(* IEC 61131-3 sources: NVM-AquaFeed-Platform/02_Software_Design/PLC/07_Implementation/Function_Blocks, 14 files *)

(* ---- FB_AlarmManager.st ---- *)
FUNCTION_BLOCK FB_AlarmManager
VAR_INPUT
    astConditions : ARRAY[0..31] OF ST_AlarmCondition;

    xAcknowledgeRequest : BOOL;
    xResetRequest : BOOL;
    udiCommandSequence : UDINT;
    uiTargetAlarmCode : UINT;
    eTargetSource : E_AlarmSource;
    usiTargetLineId : USINT;
    uiTargetDeviceId : UINT;

    udiAcceptedEventSequence : UDINT;
END_VAR
VAR_OUTPUT
    astActiveAlarms : ARRAY[0..63] OF ST_Alarm;
    stPendingEvent : ST_AlarmEvent;
    xPendingEventValid : BOOL;
    uiPendingEventCount : UINT;

    xAnyAlarmActive : BOOL;
    xAnyBlockingAlarm : BOOL;
    xAnyCriticalAlarm : BOOL;
    xAnyEmergencyAlarm : BOOL;
    eHighestSeverity : E_AlarmSeverity;
    uiActiveAlarmCount : UINT;

    xTableOverflow : BOOL;
    xEventBufferOverflow : BOOL;
    xInputRejected : BOOL;
    uiInputResultCode : UINT;

    xCommandAccepted : BOOL;
    xCommandRejected : BOOL;
    uiCommandResultCode : UINT;
    udiLastProcessedCommandSequence : UDINT;
END_VAR
VAR
    astEventBuffer : ARRAY[0..127] OF ST_AlarmEvent;
    uiEventReadIndex : UINT;
    uiEventWriteIndex : UINT;
    udiEventSequence : UDINT;
    xHasProcessedCommand : BOOL;

    iCondition : INT;
    iPreviousCondition : INT;
    iAlarm : INT;
    iFoundAlarm : INT;
    iFreeAlarm : INT;
    iCommandAlarm : INT;

    xDefinitionValid : BOOL;
    xSeverityValid : BOOL;
    xDuplicateUpdate : BOOL;
    xPolicyMatches : BOOL;
    xEmitEvent : BOOL;
    eEmitEventType : E_AlarmEventType;
END_VAR
VAR CONSTANT
    c_uiInputResultNone : UINT := 0;
    c_uiInputResultInvalidDefinition : UINT := 10;
    c_uiInputResultDuplicateKey : UINT := 11;
    c_uiInputResultPolicyChanged : UINT := 12;
    c_uiInputResultTableFull : UINT := 13;

    c_uiCommandResultNone : UINT := 0;
    c_uiCommandResultAccepted : UINT := 1;
    c_uiCommandResultConflict : UINT := 40;
    c_uiCommandResultNotFound : UINT := 41;
    c_uiCommandResultConditionActive : UINT := 42;
    c_uiCommandResultResetNotRequired : UINT := 43;
END_VAR

xCommandAccepted := FALSE;
xCommandRejected := FALSE;
uiCommandResultCode := c_uiCommandResultNone;
xInputRejected := FALSE;
uiInputResultCode := c_uiInputResultNone;

(* Desktop may remove only the exact oldest retained event. *)
IF (uiPendingEventCount > 0) AND
   (udiAcceptedEventSequence <> 0) AND
   (udiAcceptedEventSequence =
    astEventBuffer[uiEventReadIndex].EventSequence) THEN
    IF uiEventReadIndex >= 127 THEN
        uiEventReadIndex := 0;
    ELSE
        uiEventReadIndex := uiEventReadIndex + 1;
    END_IF;
    uiPendingEventCount := uiPendingEventCount - 1;
END_IF;

(* Process at most 32 explicit condition updates in array order. *)
FOR iCondition := 0 TO 31 DO
    IF astConditions[iCondition].Valid THEN
        xDuplicateUpdate := FALSE;
        IF iCondition > 0 THEN
            FOR iPreviousCondition := 0 TO iCondition - 1 DO
                IF astConditions[iPreviousCondition].Valid AND
                   (astConditions[iPreviousCondition].AlarmCode =
                    astConditions[iCondition].AlarmCode) AND
                   (astConditions[iPreviousCondition].Source =
                    astConditions[iCondition].Source) AND
                   (astConditions[iPreviousCondition].LineId =
                    astConditions[iCondition].LineId) AND
                   (astConditions[iPreviousCondition].DeviceId =
                    astConditions[iCondition].DeviceId) THEN
                    xDuplicateUpdate := TRUE;
                END_IF;
            END_FOR;
        END_IF;

        xSeverityValid := FALSE;
        CASE astConditions[iCondition].Severity OF
            ALARM_INFORMATION,
            ALARM_WARNING,
            ALARM_FAULT,
            ALARM_CRITICAL,
            ALARM_EMERGENCY:
                xSeverityValid := TRUE;
        END_CASE;

        xDefinitionValid := xSeverityValid AND
                            (astConditions[iCondition].AlarmCode >= 1000) AND
                            (astConditions[iCondition].AlarmCode <= 1999) AND
                            NOT ((astConditions[iCondition].Severity =
                                  ALARM_INFORMATION) AND
                                 astConditions[iCondition].Blocking);

        IF xDefinitionValid THEN
            CASE astConditions[iCondition].Source OF
                ALARM_SOURCE_SYSTEM:
                    xDefinitionValid :=
                        ((astConditions[iCondition].AlarmCode >= 1000) AND
                         (astConditions[iCondition].AlarmCode <= 1099)) OR
                        ((astConditions[iCondition].AlarmCode >= 1900) AND
                         (astConditions[iCondition].AlarmCode <= 1999));
                ALARM_SOURCE_COMMUNICATION:
                    xDefinitionValid :=
                        ((astConditions[iCondition].AlarmCode >= 1100) AND
                         (astConditions[iCondition].AlarmCode <= 1199)) OR
                        ((astConditions[iCondition].AlarmCode >= 1900) AND
                         (astConditions[iCondition].AlarmCode <= 1999));
                ALARM_SOURCE_SELECTOR:
                    xDefinitionValid :=
                        (astConditions[iCondition].AlarmCode >= 1200) AND
                        (astConditions[iCondition].AlarmCode <= 1299);
                ALARM_SOURCE_BLOWER:
                    xDefinitionValid :=
                        (astConditions[iCondition].AlarmCode >= 1300) AND
                        (astConditions[iCondition].AlarmCode <= 1399);
                ALARM_SOURCE_DOSING:
                    xDefinitionValid :=
                        (astConditions[iCondition].AlarmCode >= 1400) AND
                        (astConditions[iCondition].AlarmCode <= 1499);
                ALARM_SOURCE_LINE:
                    xDefinitionValid :=
                        (astConditions[iCondition].AlarmCode >= 1500) AND
                        (astConditions[iCondition].AlarmCode <= 1599);
                ALARM_SOURCE_SAFETY,
                ALARM_SOURCE_IO:
                    xDefinitionValid :=
                        ((astConditions[iCondition].AlarmCode >= 1600) AND
                         (astConditions[iCondition].AlarmCode <= 1699)) OR
                        ((astConditions[iCondition].Source =
                          ALARM_SOURCE_IO) AND
                         (astConditions[iCondition].AlarmCode >= 1900) AND
                         (astConditions[iCondition].AlarmCode <= 1999));
                ALARM_SOURCE_POWER:
                    xDefinitionValid :=
                        (astConditions[iCondition].AlarmCode >= 1700) AND
                        (astConditions[iCondition].AlarmCode <= 1799);
                ALARM_SOURCE_AUXILIARY:
                    xDefinitionValid :=
                        (astConditions[iCondition].AlarmCode >= 1800) AND
                        (astConditions[iCondition].AlarmCode <= 1899);
            ELSE
                xDefinitionValid := FALSE;
            END_CASE;
        END_IF;

        IF xDuplicateUpdate THEN
            xInputRejected := TRUE;
            uiInputResultCode := c_uiInputResultDuplicateKey;
        ELSIF NOT xDefinitionValid THEN
            xInputRejected := TRUE;
            uiInputResultCode := c_uiInputResultInvalidDefinition;
        ELSE
            iFoundAlarm := -1;
            iFreeAlarm := -1;
            FOR iAlarm := 0 TO 63 DO
                IF (astActiveAlarms[iAlarm].AlarmCode =
                    astConditions[iCondition].AlarmCode) AND
                   (astActiveAlarms[iAlarm].Source =
                    astConditions[iCondition].Source) AND
                   (astActiveAlarms[iAlarm].LineId =
                    astConditions[iCondition].LineId) AND
                   (astActiveAlarms[iAlarm].DeviceId =
                    astConditions[iCondition].DeviceId) THEN
                    iFoundAlarm := iAlarm;
                END_IF;
                IF (iFreeAlarm < 0) AND
                   (astActiveAlarms[iAlarm].State =
                    ALARM_INACTIVE) THEN
                    iFreeAlarm := iAlarm;
                END_IF;
            END_FOR;

            xEmitEvent := FALSE;

            IF astConditions[iCondition].ConditionActive THEN
                IF iFoundAlarm < 0 THEN
                    IF iFreeAlarm < 0 THEN
                        xTableOverflow := TRUE;
                        xInputRejected := TRUE;
                        uiInputResultCode :=
                            c_uiInputResultTableFull;
                    ELSE
                        IF (astActiveAlarms[iFreeAlarm].AlarmCode <>
                            astConditions[iCondition].AlarmCode) OR
                           (astActiveAlarms[iFreeAlarm].Source <>
                            astConditions[iCondition].Source) OR
                           (astActiveAlarms[iFreeAlarm].LineId <>
                            astConditions[iCondition].LineId) OR
                           (astActiveAlarms[iFreeAlarm].DeviceId <>
                            astConditions[iCondition].DeviceId) THEN
                            astActiveAlarms[iFreeAlarm].OccurrenceCount := 0;
                        END_IF;
                        iFoundAlarm := iFreeAlarm;
                    END_IF;
                END_IF;

                IF iFoundAlarm >= 0 THEN
                    xPolicyMatches :=
                        (astActiveAlarms[iFoundAlarm].State =
                         ALARM_INACTIVE) OR
                        ((astActiveAlarms[iFoundAlarm].Severity =
                          astConditions[iCondition].Severity) AND
                         (astActiveAlarms[iFoundAlarm].ResetRequired =
                          astConditions[iCondition].ResetRequired) AND
                         (astActiveAlarms[iFoundAlarm].Blocking =
                          astConditions[iCondition].Blocking));

                    IF NOT xPolicyMatches THEN
                        xInputRejected := TRUE;
                        uiInputResultCode :=
                            c_uiInputResultPolicyChanged;
                    ELSIF astActiveAlarms[iFoundAlarm].State =
                          ALARM_INACTIVE THEN
                        astActiveAlarms[iFoundAlarm].AlarmCode :=
                            astConditions[iCondition].AlarmCode;
                        astActiveAlarms[iFoundAlarm].Source :=
                            astConditions[iCondition].Source;
                        astActiveAlarms[iFoundAlarm].Severity :=
                            astConditions[iCondition].Severity;
                        astActiveAlarms[iFoundAlarm].State :=
                            ALARM_ACTIVE_UNACKNOWLEDGED;
                        astActiveAlarms[iFoundAlarm].LineId :=
                            astConditions[iCondition].LineId;
                        astActiveAlarms[iFoundAlarm].DeviceId :=
                            astConditions[iCondition].DeviceId;
                        astActiveAlarms[iFoundAlarm].ConditionActive := TRUE;
                        astActiveAlarms[iFoundAlarm].Acknowledged := FALSE;
                        astActiveAlarms[iFoundAlarm].ResetRequired :=
                            astConditions[iCondition].ResetRequired;
                        astActiveAlarms[iFoundAlarm].Blocking :=
                            astConditions[iCondition].Blocking;
                        IF astActiveAlarms[iFoundAlarm].OccurrenceCount <
                           65535 THEN
                            astActiveAlarms[iFoundAlarm].OccurrenceCount :=
                                astActiveAlarms[iFoundAlarm].OccurrenceCount + 1;
                        END_IF;
                        xEmitEvent := TRUE;
                        eEmitEventType := ALARM_EVENT_ACTIVATED;
                    ELSE
                        astActiveAlarms[iFoundAlarm].ConditionActive := TRUE;
                    END_IF;
                END_IF;
            ELSE
                IF (iFoundAlarm >= 0) AND
                   (astActiveAlarms[iFoundAlarm].State <>
                    ALARM_INACTIVE) THEN
                    xPolicyMatches :=
                        (astActiveAlarms[iFoundAlarm].Severity =
                         astConditions[iCondition].Severity) AND
                        (astActiveAlarms[iFoundAlarm].ResetRequired =
                         astConditions[iCondition].ResetRequired) AND
                        (astActiveAlarms[iFoundAlarm].Blocking =
                         astConditions[iCondition].Blocking);

                    IF NOT xPolicyMatches THEN
                        xInputRejected := TRUE;
                        uiInputResultCode :=
                            c_uiInputResultPolicyChanged;
                    ELSIF astActiveAlarms[iFoundAlarm].ConditionActive THEN
                        astActiveAlarms[iFoundAlarm].ConditionActive := FALSE;
                        IF astActiveAlarms[iFoundAlarm].ResetRequired THEN
                            astActiveAlarms[iFoundAlarm].State :=
                                ALARM_CLEARED_WAIT_RESET;
                        ELSE
                            astActiveAlarms[iFoundAlarm].State :=
                                ALARM_INACTIVE;
                            astActiveAlarms[iFoundAlarm].Acknowledged := FALSE;
                        END_IF;
                        xEmitEvent := TRUE;
                        eEmitEventType := ALARM_EVENT_CLEARED;
                    END_IF;
                END_IF;
            END_IF;

            IF xEmitEvent AND (iFoundAlarm >= 0) THEN
                IF udiEventSequence >= c_udiCounterMaximum THEN
                    xEventBufferOverflow := TRUE;
                ELSE
                    udiEventSequence := udiEventSequence + 1;
                    astActiveAlarms[iFoundAlarm].EventSequence :=
                        udiEventSequence;
                    IF eEmitEventType = ALARM_EVENT_ACTIVATED THEN
                        astActiveAlarms[iFoundAlarm].ActivationSequence :=
                            udiEventSequence;
                    END_IF;

                    IF uiPendingEventCount >=
                       c_uiAlarmEventCapacity THEN
                        xEventBufferOverflow := TRUE;
                    ELSE
                        astEventBuffer[uiEventWriteIndex].EventSequence :=
                            udiEventSequence;
                        astEventBuffer[uiEventWriteIndex].EventType :=
                            eEmitEventType;
                        astEventBuffer[uiEventWriteIndex].AlarmCode :=
                            astActiveAlarms[iFoundAlarm].AlarmCode;
                        astEventBuffer[uiEventWriteIndex].Source :=
                            astActiveAlarms[iFoundAlarm].Source;
                        astEventBuffer[uiEventWriteIndex].Severity :=
                            astActiveAlarms[iFoundAlarm].Severity;
                        astEventBuffer[uiEventWriteIndex].State :=
                            astActiveAlarms[iFoundAlarm].State;
                        astEventBuffer[uiEventWriteIndex].LineId :=
                            astActiveAlarms[iFoundAlarm].LineId;
                        astEventBuffer[uiEventWriteIndex].DeviceId :=
                            astActiveAlarms[iFoundAlarm].DeviceId;
                        IF uiEventWriteIndex >= 127 THEN
                            uiEventWriteIndex := 0;
                        ELSE
                            uiEventWriteIndex := uiEventWriteIndex + 1;
                        END_IF;
                        uiPendingEventCount := uiPendingEventCount + 1;
                    END_IF;
                END_IF;
            END_IF;
        END_IF;
    END_IF;
END_FOR;

(* Process one idempotent lifecycle command. *)
IF (xAcknowledgeRequest OR xResetRequest) AND
   (NOT xHasProcessedCommand OR
    (udiCommandSequence <>
     udiLastProcessedCommandSequence)) THEN
    udiLastProcessedCommandSequence := udiCommandSequence;
    xHasProcessedCommand := TRUE;
    iCommandAlarm := -1;

    IF xAcknowledgeRequest AND xResetRequest THEN
        xCommandRejected := TRUE;
        uiCommandResultCode := c_uiCommandResultConflict;
    ELSE
        FOR iAlarm := 0 TO 63 DO
            IF (astActiveAlarms[iAlarm].State <>
                ALARM_INACTIVE) AND
               (astActiveAlarms[iAlarm].AlarmCode =
                uiTargetAlarmCode) AND
               (astActiveAlarms[iAlarm].Source =
                eTargetSource) AND
               (astActiveAlarms[iAlarm].LineId =
                usiTargetLineId) AND
               (astActiveAlarms[iAlarm].DeviceId =
                uiTargetDeviceId) THEN
                iCommandAlarm := iAlarm;
            END_IF;
        END_FOR;

        IF iCommandAlarm < 0 THEN
            xCommandRejected := TRUE;
            uiCommandResultCode := c_uiCommandResultNotFound;
        ELSIF xAcknowledgeRequest THEN
            xCommandAccepted := TRUE;
            uiCommandResultCode := c_uiCommandResultAccepted;
            xEmitEvent := FALSE;
            IF NOT astActiveAlarms[iCommandAlarm].Acknowledged THEN
                astActiveAlarms[iCommandAlarm].Acknowledged := TRUE;
                IF astActiveAlarms[iCommandAlarm].State =
                   ALARM_ACTIVE_UNACKNOWLEDGED THEN
                    astActiveAlarms[iCommandAlarm].State :=
                        ALARM_ACTIVE_ACKNOWLEDGED;
                END_IF;
                xEmitEvent := TRUE;
                eEmitEventType := ALARM_EVENT_ACKNOWLEDGED;
            END_IF;
        ELSE
            xEmitEvent := FALSE;
            IF astActiveAlarms[iCommandAlarm].ConditionActive THEN
                xCommandRejected := TRUE;
                uiCommandResultCode :=
                    c_uiCommandResultConditionActive;
            ELSIF astActiveAlarms[iCommandAlarm].State =
                  ALARM_CLEARED_WAIT_RESET THEN
                astActiveAlarms[iCommandAlarm].State := ALARM_INACTIVE;
                astActiveAlarms[iCommandAlarm].Acknowledged := FALSE;
                xCommandAccepted := TRUE;
                uiCommandResultCode := c_uiCommandResultAccepted;
                xEmitEvent := TRUE;
                eEmitEventType := ALARM_EVENT_RESET;
            ELSE
                xCommandRejected := TRUE;
                uiCommandResultCode :=
                    c_uiCommandResultResetNotRequired;
            END_IF;
        END_IF;

        IF xEmitEvent AND (iCommandAlarm >= 0) THEN
            IF udiEventSequence >= c_udiCounterMaximum THEN
                xEventBufferOverflow := TRUE;
            ELSE
                udiEventSequence := udiEventSequence + 1;
                astActiveAlarms[iCommandAlarm].EventSequence :=
                    udiEventSequence;
                IF uiPendingEventCount >=
                   c_uiAlarmEventCapacity THEN
                    xEventBufferOverflow := TRUE;
                ELSE
                    astEventBuffer[uiEventWriteIndex].EventSequence :=
                        udiEventSequence;
                    astEventBuffer[uiEventWriteIndex].EventType :=
                        eEmitEventType;
                    astEventBuffer[uiEventWriteIndex].AlarmCode :=
                        astActiveAlarms[iCommandAlarm].AlarmCode;
                    astEventBuffer[uiEventWriteIndex].Source :=
                        astActiveAlarms[iCommandAlarm].Source;
                    astEventBuffer[uiEventWriteIndex].Severity :=
                        astActiveAlarms[iCommandAlarm].Severity;
                    astEventBuffer[uiEventWriteIndex].State :=
                        astActiveAlarms[iCommandAlarm].State;
                    astEventBuffer[uiEventWriteIndex].LineId :=
                        astActiveAlarms[iCommandAlarm].LineId;
                    astEventBuffer[uiEventWriteIndex].DeviceId :=
                        astActiveAlarms[iCommandAlarm].DeviceId;
                    IF uiEventWriteIndex >= 127 THEN
                        uiEventWriteIndex := 0;
                    ELSE
                        uiEventWriteIndex := uiEventWriteIndex + 1;
                    END_IF;
                    uiPendingEventCount := uiPendingEventCount + 1;
                END_IF;
            END_IF;
        END_IF;
    END_IF;
END_IF;

(* Recalculate bounded summaries from lifecycle records. *)
xAnyAlarmActive := FALSE;
xAnyBlockingAlarm := FALSE;
xAnyCriticalAlarm := FALSE;
xAnyEmergencyAlarm := FALSE;
eHighestSeverity := ALARM_INFORMATION;
uiActiveAlarmCount := 0;

FOR iAlarm := 0 TO 63 DO
    IF astActiveAlarms[iAlarm].State <> ALARM_INACTIVE THEN
        xAnyAlarmActive := TRUE;
        IF uiActiveAlarmCount < c_uiActiveAlarmCapacity THEN
            uiActiveAlarmCount := uiActiveAlarmCount + 1;
        END_IF;
        IF astActiveAlarms[iAlarm].Blocking THEN
            xAnyBlockingAlarm := TRUE;
        END_IF;
        IF astActiveAlarms[iAlarm].Severity > eHighestSeverity THEN
            eHighestSeverity := astActiveAlarms[iAlarm].Severity;
        END_IF;
        IF astActiveAlarms[iAlarm].Severity >= ALARM_CRITICAL THEN
            xAnyCriticalAlarm := TRUE;
        END_IF;
        IF astActiveAlarms[iAlarm].Severity = ALARM_EMERGENCY THEN
            xAnyEmergencyAlarm := TRUE;
        END_IF;
    END_IF;
END_FOR;

xPendingEventValid := uiPendingEventCount > 0;
IF xPendingEventValid THEN
    stPendingEvent := astEventBuffer[uiEventReadIndex];
ELSE
    stPendingEvent.EventSequence := 0;
    stPendingEvent.EventType := ALARM_EVENT_ACTIVATED;
    stPendingEvent.AlarmCode := 0;
    stPendingEvent.Source := ALARM_SOURCE_SYSTEM;
    stPendingEvent.Severity := ALARM_INFORMATION;
    stPendingEvent.State := ALARM_INACTIVE;
    stPendingEvent.LineId := 0;
    stPendingEvent.DeviceId := 0;
END_IF;

END_FUNCTION_BLOCK

(* ---- FB_Blower.st ---- *)
FUNCTION_BLOCK FB_Blower
VAR_INPUT
    xEnable : BOOL;
    xRunRequest : BOOL;
    xNormalStopRequest : BOOL;
    uiTargetFreqCentiHz : UINT;
    udiRequestedPostRunTimeMs : UDINT;
    udiCommandSequence : UDINT;
    udiResetSequence : UDINT;
    xSafetyOK : BOOL;
    xDriveReady : BOOL;
    xDriveRunning : BOOL;
    xDriveFault : BOOL;
    xCommunicationHealthy : BOOL;
    uiActualFreqCentiHz : UINT;
    uiDriveFaultCode : UINT;
    stConfig : ST_BlowerConfig;
    udiMonotonicTickMs : UDINT;
END_VAR
VAR_OUTPUT
    eState : E_BlowerState := BlowerDisabled;
    xDriveRunRequest : BOOL;
    uiDriveFreqCentiHz : UINT;
    xReady : BOOL;
    xRunning : BOOL;
    xAtSpeed : BOOL;
    xDosingPermitted : BOOL;
    uiDiagnosticCode : UINT;
    udiLastAcceptedSequence : UDINT;
END_VAR
VAR
    uiLatchedFreqCentiHz : UINT;
    udiLatchedPostRunTimeMs : UDINT;
    udiStateStartTickMs : UDINT;
    udiStableStartTickMs : UDINT;
    udiFeedbackLossStartTickMs : UDINT;
    udiLastResetSequence : UDINT;
    xHasAcceptedCommand : BOOL;
    xHasAcceptedReset : BOOL;
    xStableTimerActive : BOOL;
    xFeedbackLossTimerActive : BOOL;
    xConfigValid : BOOL;
    xFrequencyInTolerance : BOOL;
    diFrequencyError : DINT;
END_VAR
VAR CONSTANT
    c_uiDiagnosticNone : UINT := 0;
    c_uiDiagnosticConfig : UINT := 20;
    c_uiDiagnosticFrequencyRange : UINT := 21;
    c_uiDiagnosticDriveNotReady : UINT := 22;
    c_uiDiagnosticStartTimeout : UINT := 23;
    c_uiDiagnosticAccelerationTimeout : UINT := 24;
    c_uiDiagnosticFeedbackLoss : UINT := 25;
    c_uiDiagnosticStopTimeout : UINT := 26;
    c_uiDiagnosticCommunication : UINT := 28;
    c_uiDiagnosticDriveFault : UINT := 29;
    c_uiDiagnosticSafety : UINT := 30;
END_VAR

xDriveRunRequest := FALSE;
uiDriveFreqCentiHz := 0;
xReady := FALSE;
xRunning := FALSE;
xAtSpeed := FALSE;
xDosingPermitted := FALSE;

xConfigValid := (stConfig.uiMinimumFreqCentiHz > 0) AND
                (stConfig.uiMinimumFreqCentiHz <=
                 stConfig.uiMaximumFreqCentiHz) AND
                (stConfig.uiAtSpeedToleranceCentiHz > 0) AND
                (stConfig.udiAtSpeedStableTimeMs > 0) AND
                (stConfig.udiStartTimeoutMs > 0) AND
                (stConfig.udiAccelerationTimeoutMs > 0) AND
                (stConfig.udiFeedbackLossTimeoutMs > 0) AND
                (stConfig.udiStopTimeoutMs > 0) AND
                (stConfig.udiPostRunTimeMs > 0) AND
                (stConfig.udiMaximumPostRunTimeMs >=
                 stConfig.udiPostRunTimeMs);

diFrequencyError := UINT_TO_DINT(uiActualFreqCentiHz) -
                    UINT_TO_DINT(uiLatchedFreqCentiHz);
xFrequencyInTolerance :=
    ABS(diFrequencyError) <=
    UINT_TO_DINT(stConfig.uiAtSpeedToleranceCentiHz);

IF NOT xEnable THEN
    eState := BlowerDisabled;
    uiDiagnosticCode := c_uiDiagnosticNone;
    xStableTimerActive := FALSE;
    xFeedbackLossTimerActive := FALSE;
ELSIF NOT xSafetyOK THEN
    eState := BlowerFault;
    uiDiagnosticCode := c_uiDiagnosticSafety;
ELSIF xDriveFault THEN
    eState := BlowerFault;
    uiDiagnosticCode := c_uiDiagnosticDriveFault;
ELSIF NOT xCommunicationHealthy THEN
    eState := BlowerFault;
    uiDiagnosticCode := c_uiDiagnosticCommunication;
ELSIF NOT xConfigValid THEN
    eState := BlowerFault;
    uiDiagnosticCode := c_uiDiagnosticConfig;
ELSE
    CASE eState OF
        BlowerDisabled:
            eState := BlowerReady;
            uiDiagnosticCode := c_uiDiagnosticNone;

        BlowerReady:
            xReady := xDriveReady AND NOT xDriveRunning;

            IF xDriveRunning THEN
                eState := BlowerFault;
                uiDiagnosticCode := c_uiDiagnosticFeedbackLoss;
            ELSIF xRunRequest AND
                  (NOT xHasAcceptedCommand OR
                   (udiCommandSequence <> udiLastAcceptedSequence)) THEN
                udiLastAcceptedSequence := udiCommandSequence;
                xHasAcceptedCommand := TRUE;

                IF (uiTargetFreqCentiHz <
                    stConfig.uiMinimumFreqCentiHz) OR
                   (uiTargetFreqCentiHz >
                    stConfig.uiMaximumFreqCentiHz) OR
                   (udiRequestedPostRunTimeMs >
                    stConfig.udiMaximumPostRunTimeMs) THEN
                    uiDiagnosticCode := c_uiDiagnosticFrequencyRange;
                ELSIF NOT xDriveReady THEN
                    uiDiagnosticCode := c_uiDiagnosticDriveNotReady;
                ELSE
                    uiLatchedFreqCentiHz := uiTargetFreqCentiHz;
                    IF udiRequestedPostRunTimeMs > 0 THEN
                        udiLatchedPostRunTimeMs :=
                            udiRequestedPostRunTimeMs;
                    ELSE
                        udiLatchedPostRunTimeMs :=
                            stConfig.udiPostRunTimeMs;
                    END_IF;
                    udiStateStartTickMs := udiMonotonicTickMs;
                    xStableTimerActive := FALSE;
                    xFeedbackLossTimerActive := FALSE;
                    eState := BlowerStarting;
                    uiDiagnosticCode := c_uiDiagnosticNone;
                END_IF;
            END_IF;

        BlowerStarting:
            xDriveRunRequest := TRUE;
            uiDriveFreqCentiHz := uiLatchedFreqCentiHz;
            xRunning := xDriveRunning;

            IF xDriveRunning THEN
                udiStateStartTickMs := udiMonotonicTickMs;
                xStableTimerActive := FALSE;
                eState := BlowerAccelerating;
            ELSIF F_ElapsedMs(udiCurrentTickMs := udiMonotonicTickMs,
                             udiStartTickMs := udiStateStartTickMs) >=
                  stConfig.udiStartTimeoutMs THEN
                eState := BlowerFault;
                uiDiagnosticCode := c_uiDiagnosticStartTimeout;
            END_IF;

        BlowerAccelerating:
            xDriveRunRequest := TRUE;
            uiDriveFreqCentiHz := uiLatchedFreqCentiHz;
            xRunning := xDriveRunning;

            IF NOT xDriveRunning THEN
                eState := BlowerFault;
                uiDiagnosticCode := c_uiDiagnosticFeedbackLoss;
            ELSIF xFrequencyInTolerance THEN
                IF NOT xStableTimerActive THEN
                    udiStableStartTickMs := udiMonotonicTickMs;
                    xStableTimerActive := TRUE;
                ELSIF F_ElapsedMs(
                          udiCurrentTickMs := udiMonotonicTickMs,
                          udiStartTickMs := udiStableStartTickMs) >=
                      stConfig.udiAtSpeedStableTimeMs THEN
                    xStableTimerActive := FALSE;
                    eState := BlowerAtSpeed;
                    uiDiagnosticCode := c_uiDiagnosticNone;
                END_IF;
            ELSE
                xStableTimerActive := FALSE;
            END_IF;

            IF (eState = BlowerAccelerating) AND
               (F_ElapsedMs(udiCurrentTickMs := udiMonotonicTickMs,
                            udiStartTickMs := udiStateStartTickMs) >=
                stConfig.udiAccelerationTimeoutMs) THEN
                eState := BlowerFault;
                uiDiagnosticCode := c_uiDiagnosticAccelerationTimeout;
            END_IF;

        BlowerAtSpeed:
            xDriveRunRequest := TRUE;
            uiDriveFreqCentiHz := uiLatchedFreqCentiHz;
            xRunning := xDriveRunning;
            xAtSpeed := xDriveRunning AND xFrequencyInTolerance;
            xDosingPermitted := xAtSpeed AND xDriveReady;

            IF xNormalStopRequest OR NOT xRunRequest THEN
                udiStateStartTickMs := udiMonotonicTickMs;
                xFeedbackLossTimerActive := FALSE;
                eState := BlowerPostRun;
            ELSIF NOT xDriveRunning OR NOT xFrequencyInTolerance THEN
                IF NOT xFeedbackLossTimerActive THEN
                    udiFeedbackLossStartTickMs := udiMonotonicTickMs;
                    xFeedbackLossTimerActive := TRUE;
                ELSIF F_ElapsedMs(
                          udiCurrentTickMs := udiMonotonicTickMs,
                          udiStartTickMs := udiFeedbackLossStartTickMs) >=
                      stConfig.udiFeedbackLossTimeoutMs THEN
                    eState := BlowerFault;
                    uiDiagnosticCode := c_uiDiagnosticFeedbackLoss;
                END_IF;
            ELSE
                xFeedbackLossTimerActive := FALSE;
            END_IF;

        BlowerPostRun:
            xDriveRunRequest := TRUE;
            uiDriveFreqCentiHz := uiLatchedFreqCentiHz;
            xRunning := xDriveRunning;

            IF F_ElapsedMs(udiCurrentTickMs := udiMonotonicTickMs,
                           udiStartTickMs := udiStateStartTickMs) >=
               udiLatchedPostRunTimeMs THEN
                udiStateStartTickMs := udiMonotonicTickMs;
                eState := BlowerStopping;
            END_IF;

        BlowerStopping:
            IF NOT xDriveRunning THEN
                eState := BlowerReady;
                uiDiagnosticCode := c_uiDiagnosticNone;
            ELSIF F_ElapsedMs(udiCurrentTickMs := udiMonotonicTickMs,
                             udiStartTickMs := udiStateStartTickMs) >=
                  stConfig.udiStopTimeoutMs THEN
                eState := BlowerFault;
                uiDiagnosticCode := c_uiDiagnosticStopTimeout;
            END_IF;

        BlowerFault:
            IF (NOT xHasAcceptedReset OR
                (udiResetSequence <> udiLastResetSequence)) AND
               NOT xRunRequest AND
               NOT xNormalStopRequest AND
               xSafetyOK AND
               xCommunicationHealthy AND
               NOT xDriveFault AND
               NOT xDriveRunning AND
               xDriveReady THEN
                udiLastResetSequence := udiResetSequence;
                xHasAcceptedReset := TRUE;
                xStableTimerActive := FALSE;
                xFeedbackLossTimerActive := FALSE;
                eState := BlowerReady;
                uiDiagnosticCode := c_uiDiagnosticNone;
            END_IF;

    ELSE
        eState := BlowerFault;
        uiDiagnosticCode := c_uiDiagnosticConfig;
    END_CASE;
END_IF;

END_FUNCTION_BLOCK

(* ---- FB_CommunicationManager.st ---- *)
FUNCTION_BLOCK FB_CommunicationManager
VAR_INPUT
    xEnable : BOOL;
    uiChannelId : UINT;
    uiProfileId : UINT;
    uiChannelType : UINT;
    xRequiredForControl : BOOL;
    xTransportReady : BOOL;
    udiFreshnessTimeoutMs : UDINT;
    uiFailureThreshold : UINT;
    xRxEvent : BOOL;
    xTxEvent : BOOL;
    xProtocolErrorEvent : BOOL;
    xTimeoutEvent : BOOL;
    udiReceivedSequence : UDINT;
    udiMonotonicTickMs : UDINT;
    xResetCountersRequest : BOOL;
    udiResetSequence : UDINT;
    xServicePermission : BOOL;
END_VAR
VAR_OUTPUT
    stChannel : ST_CommunicationChannel;
    xNewFaultEvent : BOOL;
    xRecoveryEvent : BOOL;
    uiResultCode : UINT;
END_VAR
VAR
    xConfigurationValid : BOOL;
    xHasReceived : BOOL;
    xFaultLatched : BOOL;
    xWasFaultLatched : BOOL;
    xHasProcessedReset : BOOL;
    udiLastProcessedResetSequence : UDINT;
    udiElapsedSinceRxMs : UDINT;
END_VAR
VAR CONSTANT
    c_uiStateDisabled : UINT := 0;
    c_uiStateStarting : UINT := 10;
    c_uiStateReady : UINT := 20;
    c_uiStateStale : UINT := 30;
    c_uiStateFault : UINT := 90;
    c_uiDiagnosticNone : UINT := 0;
    c_uiDiagnosticConfiguration : UINT := 10;
    c_uiDiagnosticTransportUnavailable : UINT := 11;
    c_uiDiagnosticNoReceive : UINT := 12;
    c_uiDiagnosticStale : UINT := 13;
    c_uiDiagnosticFailureThreshold : UINT := 14;
    c_uiResultNone : UINT := 0;
    c_uiResultResetAccepted : UINT := 1;
    c_uiResultResetPermissionDenied : UINT := 2;
END_VAR

xNewFaultEvent := FALSE;
xRecoveryEvent := FALSE;
uiResultCode := c_uiResultNone;
xWasFaultLatched := xFaultLatched;

xConfigurationValid := (uiChannelId <> 0) AND
                       (uiProfileId <> 0) AND
                       (uiChannelType <> 0) AND
                       (udiFreshnessTimeoutMs <> 0) AND
                       (uiFailureThreshold <> 0);

stChannel.uiChannelId := uiChannelId;
stChannel.uiProfileId := uiProfileId;
stChannel.uiChannelType := uiChannelType;
stChannel.xEnabled := xEnable;
stChannel.xRequiredForControl := xRequiredForControl;
stChannel.xReady := FALSE;
stChannel.xFresh := FALSE;

IF xResetCountersRequest AND
   (NOT xHasProcessedReset OR
    (udiResetSequence <> udiLastProcessedResetSequence)) THEN
    xHasProcessedReset := TRUE;
    udiLastProcessedResetSequence := udiResetSequence;

    IF xServicePermission THEN
        stChannel.udiTxCount := 0;
        stChannel.udiRxCount := 0;
        stChannel.udiErrorCount := 0;
        stChannel.udiTimeoutCount := 0;
        stChannel.udiRetryCount := 0;
        uiResultCode := c_uiResultResetAccepted;
    ELSE
        uiResultCode := c_uiResultResetPermissionDenied;
    END_IF;
END_IF;

IF NOT xEnable THEN
    stChannel.uiState := c_uiStateDisabled;
    stChannel.uiDiagnosticCode := c_uiDiagnosticNone;
    stChannel.xFault := FALSE;
    stChannel.uiConsecutiveFailureCount := 0;
    xHasReceived := FALSE;
    xFaultLatched := FALSE;
ELSIF NOT xConfigurationValid THEN
    stChannel.uiState := c_uiStateFault;
    stChannel.uiDiagnosticCode := c_uiDiagnosticConfiguration;
    stChannel.xFault := TRUE;
    xFaultLatched := TRUE;
ELSIF NOT xTransportReady THEN
    IF xFaultLatched THEN
        stChannel.uiState := c_uiStateFault;
        stChannel.uiDiagnosticCode :=
            c_uiDiagnosticFailureThreshold;
        stChannel.xFault := TRUE;
    ELSE
        stChannel.uiState := c_uiStateStale;
        stChannel.uiDiagnosticCode :=
            c_uiDiagnosticTransportUnavailable;
        stChannel.xFault := FALSE;
    END_IF;
ELSE
    IF xTxEvent THEN
        stChannel.udiLastTxTickMs := udiMonotonicTickMs;
        IF stChannel.udiTxCount < 16#FFFFFFFF THEN
            stChannel.udiTxCount := stChannel.udiTxCount + 1;
        END_IF;
    END_IF;

    IF xProtocolErrorEvent THEN
        IF stChannel.udiErrorCount < 16#FFFFFFFF THEN
            stChannel.udiErrorCount := stChannel.udiErrorCount + 1;
        END_IF;
    END_IF;

    IF xTimeoutEvent THEN
        IF stChannel.udiErrorCount < 16#FFFFFFFF THEN
            stChannel.udiErrorCount := stChannel.udiErrorCount + 1;
        END_IF;
        IF stChannel.udiTimeoutCount < 16#FFFFFFFF THEN
            stChannel.udiTimeoutCount := stChannel.udiTimeoutCount + 1;
        END_IF;
        IF stChannel.udiRetryCount < 16#FFFFFFFF THEN
            stChannel.udiRetryCount := stChannel.udiRetryCount + 1;
        END_IF;
    END_IF;

    IF xProtocolErrorEvent OR xTimeoutEvent THEN
        IF stChannel.uiConsecutiveFailureCount < 65535 THEN
            stChannel.uiConsecutiveFailureCount :=
                stChannel.uiConsecutiveFailureCount + 1;
        END_IF;

        IF stChannel.uiConsecutiveFailureCount >=
           uiFailureThreshold THEN
            xFaultLatched := TRUE;
        END_IF;
    END_IF;

    IF xRxEvent THEN
        stChannel.udiLastRxTickMs := udiMonotonicTickMs;
        IF stChannel.udiRxCount < 16#FFFFFFFF THEN
            stChannel.udiRxCount := stChannel.udiRxCount + 1;
        END_IF;

        IF NOT xHasReceived OR
           (udiReceivedSequence <>
            stChannel.udiLastAcceptedSequence) THEN
            stChannel.udiLastAcceptedSequence :=
                udiReceivedSequence;
        END_IF;

        xHasReceived := TRUE;
        stChannel.uiConsecutiveFailureCount := 0;
        xFaultLatched := FALSE;
    END_IF;

    IF xHasReceived THEN
        udiElapsedSinceRxMs := F_ElapsedMs(
            udiCurrentTickMs := udiMonotonicTickMs,
            udiStartTickMs := stChannel.udiLastRxTickMs);
    ELSE
        udiElapsedSinceRxMs := 0;
    END_IF;

    IF xFaultLatched THEN
        stChannel.uiState := c_uiStateFault;
        stChannel.uiDiagnosticCode :=
            c_uiDiagnosticFailureThreshold;
        stChannel.xFault := TRUE;
    ELSIF NOT xHasReceived THEN
        stChannel.uiState := c_uiStateStarting;
        stChannel.uiDiagnosticCode := c_uiDiagnosticNoReceive;
        stChannel.xFault := FALSE;
    ELSIF udiElapsedSinceRxMs >= udiFreshnessTimeoutMs THEN
        stChannel.uiState := c_uiStateStale;
        stChannel.uiDiagnosticCode := c_uiDiagnosticStale;
        stChannel.xFault := FALSE;
    ELSE
        stChannel.uiState := c_uiStateReady;
        stChannel.uiDiagnosticCode := c_uiDiagnosticNone;
        stChannel.xReady := TRUE;
        stChannel.xFresh := TRUE;
        stChannel.xFault := FALSE;
    END_IF;
END_IF;

IF xFaultLatched AND NOT xWasFaultLatched THEN
    xNewFaultEvent := TRUE;
ELSIF NOT xFaultLatched AND xWasFaultLatched AND xRxEvent THEN
    xRecoveryEvent := TRUE;
END_IF;

END_FUNCTION_BLOCK

(* ---- FB_DeviceManager.st ---- *)
FUNCTION_BLOCK FB_DeviceManager
VAR_INPUT
    uiDeviceId : UINT;
    uiDeviceType : UINT;
    usiLineId : USINT;
    xEnableConfig : BOOL;
    xAutoRequest : BOOL;
    xManualRequest : BOOL;
    xRunFeedback : BOOL;
    xFaultFeedback : BOOL;
    xInterlockOK : BOOL;
    xCommunicationOK : BOOL;
END_VAR
VAR_OUTPUT
    stDevice : ST_Device;
    xReady : BOOL;
    xCommandConflict : BOOL;
    xUnexpectedRunFeedback : BOOL;
    uiDiagnosticCode : UINT;
END_VAR
VAR
    xCommonRunPermission : BOOL;
END_VAR
VAR CONSTANT
    c_uiDiagnosticNone : UINT := 0;
    c_uiDiagnosticConfiguration : UINT := 10;
    c_uiDiagnosticDisabled : UINT := 20;
    c_uiDiagnosticModeConflict : UINT := 30;
    c_uiDiagnosticEquipmentFault : UINT := 40;
    c_uiDiagnosticInterlock : UINT := 50;
    c_uiDiagnosticCommunication : UINT := 60;
END_VAR

stDevice.uiDeviceId := uiDeviceId;
stDevice.uiDeviceType := uiDeviceType;
stDevice.usiLineId := usiLineId;
stDevice.xConfigurationValid :=
    (uiDeviceId <> 0) AND (uiDeviceType <> 0);
stDevice.xEnabled :=
    stDevice.xConfigurationValid AND xEnableConfig;
stDevice.xInterlockOK := xInterlockOK;
stDevice.xCommunicationOK := xCommunicationOK;

xCommandConflict := xAutoRequest AND xManualRequest;
stDevice.xAutoMode := FALSE;
stDevice.xManualMode := FALSE;

IF stDevice.xEnabled AND NOT xCommandConflict THEN
    stDevice.xAutoMode := xAutoRequest;
    stDevice.xManualMode := xManualRequest;
END_IF;

xCommonRunPermission :=
    stDevice.xConfigurationValid AND
    stDevice.xEnabled AND
    xInterlockOK AND
    xCommunicationOK AND
    NOT xFaultFeedback;

xUnexpectedRunFeedback :=
    xRunFeedback AND NOT xCommonRunPermission;

stDevice.xUnexpectedRunFeedback :=
    xUnexpectedRunFeedback;
stDevice.xFault :=
    xFaultFeedback OR xUnexpectedRunFeedback;
stDevice.xRunning :=
    xRunFeedback AND xCommonRunPermission;
stDevice.xAvailable :=
    stDevice.xConfigurationValid AND
    stDevice.xEnabled AND
    xInterlockOK AND
    xCommunicationOK AND
    NOT stDevice.xFault;

xReady :=
    stDevice.xAvailable AND
    (stDevice.xAutoMode XOR stDevice.xManualMode) AND
    NOT xCommandConflict;

IF NOT stDevice.xConfigurationValid THEN
    uiDiagnosticCode := c_uiDiagnosticConfiguration;
ELSIF NOT stDevice.xEnabled THEN
    uiDiagnosticCode := c_uiDiagnosticDisabled;
ELSIF xCommandConflict THEN
    uiDiagnosticCode := c_uiDiagnosticModeConflict;
ELSIF xFaultFeedback THEN
    uiDiagnosticCode := c_uiDiagnosticEquipmentFault;
ELSIF NOT xInterlockOK THEN
    uiDiagnosticCode := c_uiDiagnosticInterlock;
ELSIF NOT xCommunicationOK THEN
    uiDiagnosticCode := c_uiDiagnosticCommunication;
ELSE
    uiDiagnosticCode := c_uiDiagnosticNone;
END_IF;

stDevice.uiDiagnosticCode := uiDiagnosticCode;

END_FUNCTION_BLOCK

(* ---- FB_DiagnosticsManager.st ---- *)
FUNCTION_BLOCK FB_DiagnosticsManager
VAR_INPUT
    xEnable : BOOL;
    udiScanTimeUs : UDINT;
    udiMaximumScanTimeUs : UDINT;
    xScanOverrunEvent : BOOL;
    udiScanOverrunSequence : UDINT;
    xWatchdogHealthy : BOOL;
    xConfigurationValid : BOOL;
    stIO : ST_IO;
    xRequiredCommunicationHealthy : BOOL;
    uiOfflineChannelCount : UINT;
    uiActiveAlarmCount : UINT;
    xEquipmentBlockingDiagnostic : BOOL;
    xEquipmentDegradedDiagnostic : BOOL;
    uiEquipmentDiagnosticCode : UINT;
    uiEquipmentSeverity : UINT;
    xCounterSaturation : BOOL;
END_VAR
VAR_OUTPUT
    stDiagnostics : ST_Diagnostics;
    xDiagnosticOccurrence : BOOL;
    uiOccurrenceCode : UINT;
END_VAR
VAR
    xEffectiveConfigurationValid : BOOL;
    xScanBudgetExceeded : BOOL;
    xInvalidInput : BOOL;
    xInvalidOutput : BOOL;
    xOutputMismatch : BOOL;
    xNonRequiredChannelOffline : BOOL;
    uiEquipmentSeverityBounded : UINT;
    xHasProcessedOverrun : BOOL;
    udiLastProcessedOverrunSequence : UDINT;
    xNewOverrun : BOOL;
    xInitialized : BOOL;
    xPrevConfigurationInvalid : BOOL;
    xPrevWatchdogUnhealthy : BOOL;
    xPrevRequiredIOModuleOffline : BOOL;
    xPrevInvalidInput : BOOL;
    xPrevInvalidOutput : BOOL;
    xPrevOutputMismatch : BOOL;
    xPrevRequiredCommunicationLost : BOOL;
    xPrevEquipmentBlocking : BOOL;
    xPrevScanBudgetExceeded : BOOL;
    xPrevNonRequiredChannelOffline : BOOL;
    xPrevEquipmentDegraded : BOOL;
    xPrevCounterSaturation : BOOL;
END_VAR
VAR CONSTANT
    c_uiCodeNone : UINT := 0;
    c_uiCodeConfiguration : UINT := 10;
    c_uiCodeWatchdog : UINT := 20;
    c_uiCodeRequiredIOOffline : UINT := 30;
    c_uiCodeInvalidInput : UINT := 40;
    c_uiCodeInvalidOutput : UINT := 50;
    c_uiCodeOutputMismatch : UINT := 60;
    c_uiCodeRequiredCommunication : UINT := 70;
    c_uiCodeEquipmentBlocking : UINT := 80;
    c_uiCodeScanBudget : UINT := 90;
    c_uiCodeChannelOffline : UINT := 100;
    c_uiCodeEquipmentDegraded : UINT := 110;
    c_uiCodeCounterSaturation : UINT := 120;
    c_uiSeverityWarning : UINT := 20;
    c_uiSeverityFault : UINT := 30;
    c_uiSeverityCritical : UINT := 40;
END_VAR

xDiagnosticOccurrence := FALSE;
uiOccurrenceCode := c_uiCodeNone;
xNewOverrun := FALSE;

stDiagnostics.xWatchdogHealthy := xWatchdogHealthy;
xEffectiveConfigurationValid :=
    xConfigurationValid AND
    (udiMaximumScanTimeUs <> 0);
stDiagnostics.xConfigurationValid :=
    xEffectiveConfigurationValid;
stDiagnostics.uiActiveAlarmCount := uiActiveAlarmCount;
stDiagnostics.uiInvalidInputCount := stIO.uiInvalidInputCount;
stDiagnostics.uiInvalidOutputCount := stIO.uiInvalidOutputCount;
stDiagnostics.uiOutputMismatchCount := stIO.uiOutputMismatchCount;
stDiagnostics.uiOfflineChannelCount := uiOfflineChannelCount;
stDiagnostics.udiScanTimeUs := udiScanTimeUs;

IF uiEquipmentSeverity > c_uiSeverityCritical THEN
    uiEquipmentSeverityBounded := c_uiSeverityCritical;
ELSE
    uiEquipmentSeverityBounded := uiEquipmentSeverity;
END_IF;

xScanBudgetExceeded :=
    udiScanTimeUs > udiMaximumScanTimeUs;
xInvalidInput := stIO.uiInvalidInputCount <> 0;
xInvalidOutput := stIO.uiInvalidOutputCount <> 0;
xOutputMismatch := stIO.uiOutputMismatchCount <> 0;
xNonRequiredChannelOffline :=
    (uiOfflineChannelCount <> 0) AND
    xRequiredCommunicationHealthy;

IF xEnable AND
   (udiScanTimeUs > stDiagnostics.udiMaxScanTimeUs) THEN
    stDiagnostics.udiMaxScanTimeUs := udiScanTimeUs;
END_IF;

IF xEnable AND xScanOverrunEvent AND
   (NOT xHasProcessedOverrun OR
    (udiScanOverrunSequence <>
     udiLastProcessedOverrunSequence)) THEN
    xHasProcessedOverrun := TRUE;
    udiLastProcessedOverrunSequence :=
        udiScanOverrunSequence;
    xNewOverrun := TRUE;
    IF stDiagnostics.udiScanOverrunCount <
       16#FFFFFFFF THEN
        stDiagnostics.udiScanOverrunCount :=
            stDiagnostics.udiScanOverrunCount + 1;
    END_IF;
END_IF;

stDiagnostics.xReady := FALSE;
stDiagnostics.xDegraded := FALSE;
stDiagnostics.xFault := FALSE;
stDiagnostics.uiLastDiagnosticCode := c_uiCodeNone;
stDiagnostics.uiHighestSeverity := 0;
stDiagnostics.uiActiveDiagnosticCount := 0;

IF xEnable THEN
    IF NOT xEffectiveConfigurationValid THEN
        stDiagnostics.xFault := TRUE;
        stDiagnostics.uiLastDiagnosticCode :=
            c_uiCodeConfiguration;
    ELSIF NOT xWatchdogHealthy THEN
        stDiagnostics.xFault := TRUE;
        stDiagnostics.uiLastDiagnosticCode :=
            c_uiCodeWatchdog;
    ELSIF NOT stIO.xRequiredModulesOnline THEN
        stDiagnostics.xFault := TRUE;
        stDiagnostics.uiLastDiagnosticCode :=
            c_uiCodeRequiredIOOffline;
    ELSIF xInvalidInput THEN
        stDiagnostics.xFault := TRUE;
        stDiagnostics.uiLastDiagnosticCode :=
            c_uiCodeInvalidInput;
    ELSIF xInvalidOutput THEN
        stDiagnostics.xFault := TRUE;
        stDiagnostics.uiLastDiagnosticCode :=
            c_uiCodeInvalidOutput;
    ELSIF xOutputMismatch THEN
        stDiagnostics.xFault := TRUE;
        stDiagnostics.uiLastDiagnosticCode :=
            c_uiCodeOutputMismatch;
    ELSIF NOT xRequiredCommunicationHealthy THEN
        stDiagnostics.xFault := TRUE;
        stDiagnostics.uiLastDiagnosticCode :=
            c_uiCodeRequiredCommunication;
    ELSIF xEquipmentBlockingDiagnostic THEN
        stDiagnostics.xFault := TRUE;
        IF uiEquipmentDiagnosticCode <> 0 THEN
            stDiagnostics.uiLastDiagnosticCode :=
                uiEquipmentDiagnosticCode;
        ELSE
            stDiagnostics.uiLastDiagnosticCode :=
                c_uiCodeEquipmentBlocking;
        END_IF;
    ELSIF xScanBudgetExceeded THEN
        stDiagnostics.xDegraded := TRUE;
        stDiagnostics.uiLastDiagnosticCode :=
            c_uiCodeScanBudget;
    ELSIF xNonRequiredChannelOffline THEN
        stDiagnostics.xDegraded := TRUE;
        stDiagnostics.uiLastDiagnosticCode :=
            c_uiCodeChannelOffline;
    ELSIF xEquipmentDegradedDiagnostic THEN
        stDiagnostics.xDegraded := TRUE;
        IF uiEquipmentDiagnosticCode <> 0 THEN
            stDiagnostics.uiLastDiagnosticCode :=
                uiEquipmentDiagnosticCode;
        ELSE
            stDiagnostics.uiLastDiagnosticCode :=
                c_uiCodeEquipmentDegraded;
        END_IF;
    ELSIF xCounterSaturation THEN
        stDiagnostics.xDegraded := TRUE;
        stDiagnostics.uiLastDiagnosticCode :=
            c_uiCodeCounterSaturation;
    ELSE
        stDiagnostics.xReady := TRUE;
    END_IF;

    IF stDiagnostics.xFault THEN
        IF NOT xWatchdogHealthy THEN
            stDiagnostics.uiHighestSeverity :=
                c_uiSeverityCritical;
        ELSIF xEquipmentBlockingDiagnostic AND
              (uiEquipmentSeverityBounded >
               c_uiSeverityFault) THEN
            stDiagnostics.uiHighestSeverity :=
                uiEquipmentSeverityBounded;
        ELSE
            stDiagnostics.uiHighestSeverity :=
                c_uiSeverityFault;
        END_IF;
    ELSIF stDiagnostics.xDegraded THEN
        IF xEquipmentDegradedDiagnostic AND
           (uiEquipmentSeverityBounded >
            c_uiSeverityWarning) THEN
            stDiagnostics.uiHighestSeverity :=
                uiEquipmentSeverityBounded;
        ELSE
            stDiagnostics.uiHighestSeverity :=
                c_uiSeverityWarning;
        END_IF;
    END_IF;

    IF NOT xEffectiveConfigurationValid THEN
        stDiagnostics.uiActiveDiagnosticCount :=
            stDiagnostics.uiActiveDiagnosticCount + 1;
    END_IF;
    IF NOT xWatchdogHealthy THEN
        stDiagnostics.uiActiveDiagnosticCount :=
            stDiagnostics.uiActiveDiagnosticCount + 1;
    END_IF;
    IF NOT stIO.xRequiredModulesOnline THEN
        stDiagnostics.uiActiveDiagnosticCount :=
            stDiagnostics.uiActiveDiagnosticCount + 1;
    END_IF;
    IF xInvalidInput THEN
        stDiagnostics.uiActiveDiagnosticCount :=
            stDiagnostics.uiActiveDiagnosticCount + 1;
    END_IF;
    IF xInvalidOutput THEN
        stDiagnostics.uiActiveDiagnosticCount :=
            stDiagnostics.uiActiveDiagnosticCount + 1;
    END_IF;
    IF xOutputMismatch THEN
        stDiagnostics.uiActiveDiagnosticCount :=
            stDiagnostics.uiActiveDiagnosticCount + 1;
    END_IF;
    IF NOT xRequiredCommunicationHealthy THEN
        stDiagnostics.uiActiveDiagnosticCount :=
            stDiagnostics.uiActiveDiagnosticCount + 1;
    END_IF;
    IF xEquipmentBlockingDiagnostic THEN
        stDiagnostics.uiActiveDiagnosticCount :=
            stDiagnostics.uiActiveDiagnosticCount + 1;
    END_IF;
    IF xScanBudgetExceeded THEN
        stDiagnostics.uiActiveDiagnosticCount :=
            stDiagnostics.uiActiveDiagnosticCount + 1;
    END_IF;
    IF xNonRequiredChannelOffline THEN
        stDiagnostics.uiActiveDiagnosticCount :=
            stDiagnostics.uiActiveDiagnosticCount + 1;
    END_IF;
    IF xEquipmentDegradedDiagnostic THEN
        stDiagnostics.uiActiveDiagnosticCount :=
            stDiagnostics.uiActiveDiagnosticCount + 1;
    END_IF;
    IF xCounterSaturation THEN
        stDiagnostics.uiActiveDiagnosticCount :=
            stDiagnostics.uiActiveDiagnosticCount + 1;
    END_IF;

    IF xInitialized THEN
        IF NOT xEffectiveConfigurationValid AND
           NOT xPrevConfigurationInvalid THEN
            uiOccurrenceCode := c_uiCodeConfiguration;
        ELSIF NOT xWatchdogHealthy AND
              NOT xPrevWatchdogUnhealthy THEN
            uiOccurrenceCode := c_uiCodeWatchdog;
        ELSIF NOT stIO.xRequiredModulesOnline AND
              NOT xPrevRequiredIOModuleOffline THEN
            uiOccurrenceCode := c_uiCodeRequiredIOOffline;
        ELSIF xInvalidInput AND NOT xPrevInvalidInput THEN
            uiOccurrenceCode := c_uiCodeInvalidInput;
        ELSIF xInvalidOutput AND NOT xPrevInvalidOutput THEN
            uiOccurrenceCode := c_uiCodeInvalidOutput;
        ELSIF xOutputMismatch AND NOT xPrevOutputMismatch THEN
            uiOccurrenceCode := c_uiCodeOutputMismatch;
        ELSIF NOT xRequiredCommunicationHealthy AND
              NOT xPrevRequiredCommunicationLost THEN
            uiOccurrenceCode :=
                c_uiCodeRequiredCommunication;
        ELSIF xEquipmentBlockingDiagnostic AND
              NOT xPrevEquipmentBlocking THEN
            IF uiEquipmentDiagnosticCode <> 0 THEN
                uiOccurrenceCode :=
                    uiEquipmentDiagnosticCode;
            ELSE
                uiOccurrenceCode :=
                    c_uiCodeEquipmentBlocking;
            END_IF;
        ELSIF xNewOverrun OR
              (xScanBudgetExceeded AND
               NOT xPrevScanBudgetExceeded) THEN
            uiOccurrenceCode := c_uiCodeScanBudget;
        ELSIF xNonRequiredChannelOffline AND
              NOT xPrevNonRequiredChannelOffline THEN
            uiOccurrenceCode := c_uiCodeChannelOffline;
        ELSIF xEquipmentDegradedDiagnostic AND
              NOT xPrevEquipmentDegraded THEN
            IF uiEquipmentDiagnosticCode <> 0 THEN
                uiOccurrenceCode :=
                    uiEquipmentDiagnosticCode;
            ELSE
                uiOccurrenceCode :=
                    c_uiCodeEquipmentDegraded;
            END_IF;
        ELSIF xCounterSaturation AND
              NOT xPrevCounterSaturation THEN
            uiOccurrenceCode :=
                c_uiCodeCounterSaturation;
        END_IF;
    END_IF;

    IF uiOccurrenceCode <> c_uiCodeNone THEN
        xDiagnosticOccurrence := TRUE;
        IF stDiagnostics.udiDiagnosticOccurrenceCount <
           16#FFFFFFFF THEN
            stDiagnostics.udiDiagnosticOccurrenceCount :=
                stDiagnostics.udiDiagnosticOccurrenceCount + 1;
        END_IF;
    END_IF;

    xInitialized := TRUE;
ELSE
    xInitialized := FALSE;
END_IF;

xPrevConfigurationInvalid := NOT xEffectiveConfigurationValid;
xPrevWatchdogUnhealthy := NOT xWatchdogHealthy;
xPrevRequiredIOModuleOffline :=
    NOT stIO.xRequiredModulesOnline;
xPrevInvalidInput := xInvalidInput;
xPrevInvalidOutput := xInvalidOutput;
xPrevOutputMismatch := xOutputMismatch;
xPrevRequiredCommunicationLost :=
    NOT xRequiredCommunicationHealthy;
xPrevEquipmentBlocking :=
    xEquipmentBlockingDiagnostic;
xPrevScanBudgetExceeded := xScanBudgetExceeded;
xPrevNonRequiredChannelOffline :=
    xNonRequiredChannelOffline;
xPrevEquipmentDegraded :=
    xEquipmentDegradedDiagnostic;
xPrevCounterSaturation := xCounterSaturation;

END_FUNCTION_BLOCK

(* ---- FB_Dosing.st ---- *)
FUNCTION_BLOCK FB_Dosing
VAR_INPUT
    xEnable : BOOL;
    xStartRequest : BOOL;
    xStopRequest : BOOL;
    udiCommandSequence : UDINT;
    udiResetSequence : UDINT;
    udiJobId : UDINT;
    uiOutletId : UINT;
    udiTargetCentiKg : UDINT;
    uiTargetSpeedPermille : UINT;
    udiCentiKgPer1000Pulses : UDINT;
    uiCalibrationVersion : UINT;
    xSelectorInPosition : BOOL;
    xBlowerAtSpeed : BOOL;
    xFeedAvailable : BOOL;
    xSafetyOK : BOOL;
    xDriveRunning : BOOL;
    xDriveFault : BOOL;
    xPulse : BOOL;
    stConfig : ST_DosingConfig;
    udiMonotonicTickMs : UDINT;
END_VAR
VAR_OUTPUT
    eState : E_DosingState := DosingDisabled;
    xMotorRunRequest : BOOL;
    uiSpeedPermille : UINT;
    xReady : BOOL;
    xRunning : BOOL;
    xFault : BOOL;
    xCompletedEvent : BOOL;
    udiDeliveredCentiKg : UDINT;
    udiDeliveredIncrementCentiKg : UDINT;
    uiDiagnosticCode : UINT;
    udiLastAcceptedSequence : UDINT;
END_VAR
VAR
    udiLatchedJobId : UDINT;
    uiLatchedOutletId : UINT;
    udiLatchedTargetCentiKg : UDINT;
    uiLatchedSpeedPermille : UINT;
    udiLatchedCentiKgPer1000Pulses : UDINT;
    uiLatchedCalibrationVersion : UINT;
    udiTransactionStartTickMs : UDINT;
    udiStateStartTickMs : UDINT;
    udiLastPulseTickMs : UDINT;
    udiPulseRemainder : UDINT;
    udiBaseIncrement : UDINT;
    udiRemainderStep : UDINT;
    udiPulseIncrement : UDINT;
    udiLastResetSequence : UDINT;
    xHasAcceptedCommand : BOOL;
    xHasAcceptedReset : BOOL;
    xCompletionPending : BOOL;
    xConfigValid : BOOL;
    xTransactionActive : BOOL;
    xParameterChanged : BOOL;
    xTargetReached : BOOL;
END_VAR
VAR CONSTANT
    c_uiDiagnosticNone : UINT := 0;
    c_uiDiagnosticConfig : UINT := 40;
    c_uiDiagnosticInvalidCommand : UINT := 41;
    c_uiDiagnosticInterlock : UINT := 42;
    c_uiDiagnosticDriveFault : UINT := 43;
    c_uiDiagnosticStartTimeout : UINT := 44;
    c_uiDiagnosticFirstPulseTimeout : UINT := 45;
    c_uiDiagnosticNoFlow : UINT := 46;
    c_uiDiagnosticExcessiveRate : UINT := 47;
    c_uiDiagnosticTargetTimeout : UINT := 48;
    c_uiDiagnosticStopTimeout : UINT := 49;
    c_uiDiagnosticUnexpectedPulse : UINT := 50;
    c_uiDiagnosticParameterChanged : UINT := 51;
    c_uiDiagnosticArithmetic : UINT := 52;
    c_uiDiagnosticFeedback : UINT := 53;
    c_uiDiagnosticStopped : UINT := 54;
END_VAR

xMotorRunRequest := FALSE;
uiSpeedPermille := 0;
xReady := FALSE;
xRunning := FALSE;
xFault := FALSE;
xCompletedEvent := FALSE;
udiDeliveredIncrementCentiKg := 0;
udiPulseIncrement := 0;

xConfigValid := (stConfig.udiMaximumTargetCentiKg > 0) AND
                (stConfig.udiMaximumCentiKgPer1000Pulses > 0) AND
                (stConfig.uiMinimumSpeedPermille > 0) AND
                (stConfig.uiMinimumSpeedPermille <= 1000) AND
                (stConfig.udiStartTimeoutMs > 0) AND
                (stConfig.udiFirstPulseTimeoutMs > 0) AND
                (stConfig.udiNoFlowTimeoutMs > 0) AND
                (stConfig.udiMinimumPulseIntervalMs > 0) AND
                (stConfig.udiTargetTimeoutMs > 0) AND
                (stConfig.udiStopTimeoutMs > 0);

xTransactionActive := (eState = DosingStarting) OR
                      (eState = DosingWaitFirstPulse) OR
                      (eState = DosingActive) OR
                      (eState = DosingStopping);

xParameterChanged := xTransactionActive AND
    ((udiJobId <> udiLatchedJobId) OR
     (uiOutletId <> uiLatchedOutletId) OR
     (udiTargetCentiKg <> udiLatchedTargetCentiKg) OR
     (uiTargetSpeedPermille <> uiLatchedSpeedPermille) OR
     (udiCentiKgPer1000Pulses <>
      udiLatchedCentiKgPer1000Pulses) OR
     (uiCalibrationVersion <> uiLatchedCalibrationVersion));

IF NOT xEnable THEN
    eState := DosingDisabled;
    uiDiagnosticCode := c_uiDiagnosticNone;
    xCompletionPending := FALSE;
ELSIF NOT xConfigValid THEN
    eState := DosingFault;
    uiDiagnosticCode := c_uiDiagnosticConfig;
ELSIF xDriveFault THEN
    eState := DosingFault;
    uiDiagnosticCode := c_uiDiagnosticDriveFault;
ELSIF xTransactionActive AND
      (NOT xSafetyOK OR
       NOT xSelectorInPosition OR
       NOT xBlowerAtSpeed OR
       NOT xFeedAvailable) THEN
    eState := DosingFault;
    uiDiagnosticCode := c_uiDiagnosticInterlock;
ELSIF ((eState = DosingWaitFirstPulse) OR
       (eState = DosingActive)) AND
      NOT xDriveRunning THEN
    eState := DosingFault;
    uiDiagnosticCode := c_uiDiagnosticFeedback;
ELSE
    IF xParameterChanged THEN
        uiDiagnosticCode := c_uiDiagnosticParameterChanged;
    END_IF;

    CASE eState OF
        DosingDisabled:
            eState := DosingReady;
            udiDeliveredCentiKg := 0;
            uiDiagnosticCode := c_uiDiagnosticNone;

        DosingReady:
            xReady := TRUE;

            IF xPulse THEN
                uiDiagnosticCode := c_uiDiagnosticUnexpectedPulse;
            END_IF;

            IF xStartRequest AND
               (NOT xHasAcceptedCommand OR
                (udiCommandSequence <> udiLastAcceptedSequence)) THEN
                udiLastAcceptedSequence := udiCommandSequence;
                xHasAcceptedCommand := TRUE;

                IF (udiJobId = 0) OR
                   (uiOutletId = 0) OR
                   (uiCalibrationVersion = 0) OR
                   (udiTargetCentiKg = 0) OR
                   (udiTargetCentiKg >
                    stConfig.udiMaximumTargetCentiKg) OR
                   (stConfig.udiCompletionToleranceCentiKg >=
                    udiTargetCentiKg) OR
                   (uiTargetSpeedPermille <
                    stConfig.uiMinimumSpeedPermille) OR
                   (uiTargetSpeedPermille > 1000) OR
                   (udiCentiKgPer1000Pulses = 0) OR
                   (udiCentiKgPer1000Pulses >
                    stConfig.udiMaximumCentiKgPer1000Pulses) THEN
                    uiDiagnosticCode := c_uiDiagnosticInvalidCommand;
                ELSIF NOT xSafetyOK OR
                      NOT xSelectorInPosition OR
                      NOT xBlowerAtSpeed OR
                      NOT xFeedAvailable OR
                      xDriveRunning THEN
                    uiDiagnosticCode := c_uiDiagnosticInterlock;
                ELSE
                    udiLatchedJobId := udiJobId;
                    uiLatchedOutletId := uiOutletId;
                    udiLatchedTargetCentiKg := udiTargetCentiKg;
                    uiLatchedSpeedPermille := uiTargetSpeedPermille;
                    udiLatchedCentiKgPer1000Pulses :=
                        udiCentiKgPer1000Pulses;
                    uiLatchedCalibrationVersion :=
                        uiCalibrationVersion;
                    udiDeliveredCentiKg := 0;
                    udiPulseRemainder := 0;
                    udiTransactionStartTickMs :=
                        udiMonotonicTickMs;
                    udiStateStartTickMs := udiMonotonicTickMs;
                    xCompletionPending := FALSE;
                    eState := DosingStarting;
                    uiDiagnosticCode := c_uiDiagnosticNone;
                END_IF;
            END_IF;

        DosingStarting:
            xMotorRunRequest := TRUE;
            uiSpeedPermille := uiLatchedSpeedPermille;
            xRunning := xDriveRunning;

            IF xStopRequest THEN
                xMotorRunRequest := FALSE;
                uiSpeedPermille := 0;
                udiStateStartTickMs := udiMonotonicTickMs;
                xCompletionPending := FALSE;
                eState := DosingStopping;
                uiDiagnosticCode := c_uiDiagnosticStopped;
            ELSIF xDriveRunning THEN
                udiStateStartTickMs := udiMonotonicTickMs;
                eState := DosingWaitFirstPulse;
            ELSIF F_ElapsedMs(udiCurrentTickMs := udiMonotonicTickMs,
                             udiStartTickMs := udiStateStartTickMs) >=
                  stConfig.udiStartTimeoutMs THEN
                eState := DosingFault;
                uiDiagnosticCode := c_uiDiagnosticStartTimeout;
            END_IF;

        DosingWaitFirstPulse:
            xMotorRunRequest := TRUE;
            uiSpeedPermille := uiLatchedSpeedPermille;
            xRunning := TRUE;

            IF xStopRequest THEN
                xMotorRunRequest := FALSE;
                uiSpeedPermille := 0;
                udiStateStartTickMs := udiMonotonicTickMs;
                xCompletionPending := FALSE;
                eState := DosingStopping;
                uiDiagnosticCode := c_uiDiagnosticStopped;
            ELSIF xPulse THEN
                udiBaseIncrement :=
                    udiLatchedCentiKgPer1000Pulses / 1000;
                udiRemainderStep :=
                    udiLatchedCentiKgPer1000Pulses MOD 1000;
                udiPulseIncrement := udiBaseIncrement;
                udiPulseRemainder :=
                    udiPulseRemainder + udiRemainderStep;

                IF udiPulseRemainder >= 1000 THEN
                    udiPulseRemainder := udiPulseRemainder - 1000;
                    udiPulseIncrement := udiPulseIncrement + 1;
                END_IF;

                IF (udiPulseIncrement >
                    stConfig.udiMaximumTargetCentiKg) OR
                   (udiDeliveredCentiKg >
                    (stConfig.udiMaximumTargetCentiKg -
                     udiPulseIncrement)) THEN
                    udiDeliveredCentiKg :=
                        stConfig.udiMaximumTargetCentiKg;
                    eState := DosingFault;
                    uiDiagnosticCode := c_uiDiagnosticArithmetic;
                ELSE
                    udiDeliveredCentiKg :=
                        udiDeliveredCentiKg + udiPulseIncrement;
                    udiDeliveredIncrementCentiKg :=
                        udiPulseIncrement;
                    udiLastPulseTickMs := udiMonotonicTickMs;

                    xTargetReached :=
                        (udiDeliveredCentiKg >=
                         udiLatchedTargetCentiKg) OR
                        ((udiLatchedTargetCentiKg >
                          udiDeliveredCentiKg) AND
                         ((udiLatchedTargetCentiKg -
                           udiDeliveredCentiKg) <=
                          stConfig.udiCompletionToleranceCentiKg));

                    IF xTargetReached THEN
                        xMotorRunRequest := FALSE;
                        uiSpeedPermille := 0;
                        udiStateStartTickMs := udiMonotonicTickMs;
                        xCompletionPending := TRUE;
                        eState := DosingStopping;
                    ELSE
                        eState := DosingActive;
                    END_IF;
                END_IF;
            ELSIF F_ElapsedMs(
                      udiCurrentTickMs := udiMonotonicTickMs,
                      udiStartTickMs := udiStateStartTickMs) >=
                  stConfig.udiFirstPulseTimeoutMs THEN
                eState := DosingFault;
                uiDiagnosticCode := c_uiDiagnosticFirstPulseTimeout;
            END_IF;

        DosingActive:
            xMotorRunRequest := TRUE;
            uiSpeedPermille := uiLatchedSpeedPermille;
            xRunning := TRUE;

            IF xStopRequest THEN
                xMotorRunRequest := FALSE;
                uiSpeedPermille := 0;
                udiStateStartTickMs := udiMonotonicTickMs;
                xCompletionPending := FALSE;
                eState := DosingStopping;
                uiDiagnosticCode := c_uiDiagnosticStopped;
            ELSIF xPulse THEN
                IF F_ElapsedMs(
                       udiCurrentTickMs := udiMonotonicTickMs,
                       udiStartTickMs := udiLastPulseTickMs) <
                   stConfig.udiMinimumPulseIntervalMs THEN
                    eState := DosingFault;
                    uiDiagnosticCode := c_uiDiagnosticExcessiveRate;
                ELSE
                    udiBaseIncrement :=
                        udiLatchedCentiKgPer1000Pulses / 1000;
                    udiRemainderStep :=
                        udiLatchedCentiKgPer1000Pulses MOD 1000;
                    udiPulseIncrement := udiBaseIncrement;
                    udiPulseRemainder :=
                        udiPulseRemainder + udiRemainderStep;

                    IF udiPulseRemainder >= 1000 THEN
                        udiPulseRemainder :=
                            udiPulseRemainder - 1000;
                        udiPulseIncrement := udiPulseIncrement + 1;
                    END_IF;

                    IF (udiPulseIncrement >
                        stConfig.udiMaximumTargetCentiKg) OR
                       (udiDeliveredCentiKg >
                        (stConfig.udiMaximumTargetCentiKg -
                         udiPulseIncrement)) THEN
                        udiDeliveredCentiKg :=
                            stConfig.udiMaximumTargetCentiKg;
                        eState := DosingFault;
                        uiDiagnosticCode := c_uiDiagnosticArithmetic;
                    ELSE
                        udiDeliveredCentiKg :=
                            udiDeliveredCentiKg +
                            udiPulseIncrement;
                        udiDeliveredIncrementCentiKg :=
                            udiPulseIncrement;
                        udiLastPulseTickMs := udiMonotonicTickMs;
                    END_IF;
                END_IF;
            ELSIF F_ElapsedMs(
                      udiCurrentTickMs := udiMonotonicTickMs,
                      udiStartTickMs := udiLastPulseTickMs) >=
                  stConfig.udiNoFlowTimeoutMs THEN
                eState := DosingFault;
                uiDiagnosticCode := c_uiDiagnosticNoFlow;
            END_IF;

            xTargetReached :=
                (udiDeliveredCentiKg >=
                 udiLatchedTargetCentiKg) OR
                ((udiLatchedTargetCentiKg >
                  udiDeliveredCentiKg) AND
                 ((udiLatchedTargetCentiKg -
                   udiDeliveredCentiKg) <=
                  stConfig.udiCompletionToleranceCentiKg));

            IF (eState = DosingActive) AND xTargetReached THEN
                xMotorRunRequest := FALSE;
                uiSpeedPermille := 0;
                udiStateStartTickMs := udiMonotonicTickMs;
                xCompletionPending := TRUE;
                eState := DosingStopping;
            ELSIF (eState = DosingActive) AND
                  (F_ElapsedMs(
                       udiCurrentTickMs := udiMonotonicTickMs,
                       udiStartTickMs := udiTransactionStartTickMs) >=
                   stConfig.udiTargetTimeoutMs) THEN
                eState := DosingFault;
                uiDiagnosticCode := c_uiDiagnosticTargetTimeout;
            END_IF;

        DosingStopping:
            IF NOT xDriveRunning THEN
                IF xCompletionPending THEN
                    eState := DosingComplete;
                ELSE
                    eState := DosingReady;
                END_IF;
            ELSIF F_ElapsedMs(udiCurrentTickMs := udiMonotonicTickMs,
                             udiStartTickMs := udiStateStartTickMs) >=
                  stConfig.udiStopTimeoutMs THEN
                eState := DosingFault;
                uiDiagnosticCode := c_uiDiagnosticStopTimeout;
            END_IF;

        DosingComplete:
            xCompletedEvent := TRUE;
            xCompletionPending := FALSE;
            eState := DosingReady;
            uiDiagnosticCode := c_uiDiagnosticNone;

        DosingFault:
            xFault := TRUE;

            IF (NOT xHasAcceptedReset OR
                (udiResetSequence <> udiLastResetSequence)) AND
               NOT xStartRequest AND
               NOT xDriveRunning AND
               NOT xDriveFault AND
               xSafetyOK AND
               xSelectorInPosition AND
               xBlowerAtSpeed AND
               xFeedAvailable THEN
                udiLastResetSequence := udiResetSequence;
                xHasAcceptedReset := TRUE;
                xCompletionPending := FALSE;
                eState := DosingReady;
                uiDiagnosticCode := c_uiDiagnosticNone;
            END_IF;

    ELSE
        eState := DosingFault;
        uiDiagnosticCode := c_uiDiagnosticConfig;
    END_CASE;
END_IF;

IF eState = DosingFault THEN
    xMotorRunRequest := FALSE;
    uiSpeedPermille := 0;
    xRunning := FALSE;
    xFault := TRUE;
    xCompletedEvent := FALSE;
END_IF;

END_FUNCTION_BLOCK

(* ---- FB_HealthMonitor.st ---- *)
FUNCTION_BLOCK FB_HealthMonitor
VAR_INPUT
    xSystemOperational : BOOL;
    xSafetyHealthy : BOOL;
    xIOHealthy : BOOL;
    xRequiredCommunicationHealthy : BOOL;
    xDesktopCommunicationHealthy : BOOL;
    xSelectorHealthy : BOOL;
    xBlowerHealthy : BOOL;
    xDosingHealthy : BOOL;
    xConfigurationValid : BOOL;
    xDiagnosticsBlocking : BOOL;
    xDiagnosticsDegraded : BOOL;
    uiDiagnosticsSeverity : UINT;
END_VAR
VAR_OUTPUT
    stHealth : ST_HealthStatus;
    xTransitionEvent : BOOL;
    uiTransitionCode : UINT;
END_VAR
VAR
    stPrevious : ST_HealthStatus;
    xInitialized : BOOL;
    xMaterialChange : BOOL;
    uiBoundedDiagnosticSeverity : UINT;
END_VAR
VAR CONSTANT
    c_uiReasonNone : UINT := 0;
    c_uiReasonSafety : UINT := 10;
    c_uiReasonConfiguration : UINT := 20;
    c_uiReasonIO : UINT := 30;
    c_uiReasonSystem : UINT := 40;
    c_uiReasonRequiredCommunication : UINT := 50;
    c_uiReasonSelector : UINT := 60;
    c_uiReasonBlower : UINT := 70;
    c_uiReasonDosing : UINT := 80;
    c_uiReasonDiagnostics : UINT := 90;
    c_uiReasonDesktopCommunication : UINT := 100;
    c_uiReasonDiagnosticsDegraded : UINT := 110;
    c_uiSeverityWarning : UINT := 20;
    c_uiSeverityFault : UINT := 30;
    c_uiSeverityCritical : UINT := 40;
END_VAR

xTransitionEvent := FALSE;
stHealth.xSafetyHealthy := xSafetyHealthy;
stHealth.xIOHealthy := xIOHealthy;
stHealth.xRequiredCommunicationHealthy :=
    xRequiredCommunicationHealthy;
stHealth.xSelectorHealthy := xSelectorHealthy;
stHealth.xBlowerHealthy := xBlowerHealthy;
stHealth.xDosingHealthy := xDosingHealthy;
stHealth.xConfigurationValid := xConfigurationValid;

IF uiDiagnosticsSeverity > c_uiSeverityCritical THEN
    uiBoundedDiagnosticSeverity := c_uiSeverityCritical;
ELSE
    uiBoundedDiagnosticSeverity := uiDiagnosticsSeverity;
END_IF;

stHealth.xBlockingFault := FALSE;
stHealth.uiBlockingReasonCode := c_uiReasonNone;

IF NOT xSafetyHealthy THEN
    stHealth.xBlockingFault := TRUE;
    stHealth.uiBlockingReasonCode := c_uiReasonSafety;
ELSIF NOT xConfigurationValid THEN
    stHealth.xBlockingFault := TRUE;
    stHealth.uiBlockingReasonCode := c_uiReasonConfiguration;
ELSIF NOT xIOHealthy THEN
    stHealth.xBlockingFault := TRUE;
    stHealth.uiBlockingReasonCode := c_uiReasonIO;
ELSIF NOT xSystemOperational THEN
    stHealth.xBlockingFault := TRUE;
    stHealth.uiBlockingReasonCode := c_uiReasonSystem;
ELSIF NOT xRequiredCommunicationHealthy THEN
    stHealth.xBlockingFault := TRUE;
    stHealth.uiBlockingReasonCode :=
        c_uiReasonRequiredCommunication;
ELSIF NOT xSelectorHealthy THEN
    stHealth.xBlockingFault := TRUE;
    stHealth.uiBlockingReasonCode := c_uiReasonSelector;
ELSIF NOT xBlowerHealthy THEN
    stHealth.xBlockingFault := TRUE;
    stHealth.uiBlockingReasonCode := c_uiReasonBlower;
ELSIF NOT xDosingHealthy THEN
    stHealth.xBlockingFault := TRUE;
    stHealth.uiBlockingReasonCode := c_uiReasonDosing;
ELSIF xDiagnosticsBlocking THEN
    stHealth.xBlockingFault := TRUE;
    stHealth.uiBlockingReasonCode := c_uiReasonDiagnostics;
END_IF;

stHealth.xReadyForNewJob :=
    NOT stHealth.xBlockingFault AND
    xDesktopCommunicationHealthy;
stHealth.xCurrentJobMayContinue :=
    NOT stHealth.xBlockingFault;

stHealth.xDegraded :=
    NOT stHealth.xBlockingFault AND
    (NOT xDesktopCommunicationHealthy OR
     xDiagnosticsDegraded);
stHealth.uiDegradedReasonCode := c_uiReasonNone;

IF stHealth.xDegraded THEN
    IF NOT xDesktopCommunicationHealthy THEN
        stHealth.uiDegradedReasonCode :=
            c_uiReasonDesktopCommunication;
    ELSE
        stHealth.uiDegradedReasonCode :=
            c_uiReasonDiagnosticsDegraded;
    END_IF;
END_IF;

IF stHealth.xBlockingFault THEN
    IF stHealth.uiBlockingReasonCode = c_uiReasonSafety THEN
        stHealth.uiHighestSeverity := c_uiSeverityCritical;
    ELSIF uiBoundedDiagnosticSeverity >
          c_uiSeverityFault THEN
        stHealth.uiHighestSeverity :=
            uiBoundedDiagnosticSeverity;
    ELSE
        stHealth.uiHighestSeverity := c_uiSeverityFault;
    END_IF;
ELSIF stHealth.xDegraded THEN
    IF uiBoundedDiagnosticSeverity >
       c_uiSeverityWarning THEN
        stHealth.uiHighestSeverity :=
            uiBoundedDiagnosticSeverity;
    ELSE
        stHealth.uiHighestSeverity :=
            c_uiSeverityWarning;
    END_IF;
ELSE
    stHealth.uiHighestSeverity := 0;
END_IF;

IF stHealth.xBlockingFault THEN
    uiTransitionCode := stHealth.uiBlockingReasonCode;
ELSE
    uiTransitionCode := stHealth.uiDegradedReasonCode;
END_IF;

xMaterialChange :=
    (stHealth.xReadyForNewJob <>
     stPrevious.xReadyForNewJob) OR
    (stHealth.xCurrentJobMayContinue <>
     stPrevious.xCurrentJobMayContinue) OR
    (stHealth.xDegraded <> stPrevious.xDegraded) OR
    (stHealth.xBlockingFault <>
     stPrevious.xBlockingFault) OR
    (stHealth.xSafetyHealthy <>
     stPrevious.xSafetyHealthy) OR
    (stHealth.xIOHealthy <> stPrevious.xIOHealthy) OR
    (stHealth.xRequiredCommunicationHealthy <>
     stPrevious.xRequiredCommunicationHealthy) OR
    (stHealth.xSelectorHealthy <>
     stPrevious.xSelectorHealthy) OR
    (stHealth.xBlowerHealthy <>
     stPrevious.xBlowerHealthy) OR
    (stHealth.xDosingHealthy <>
     stPrevious.xDosingHealthy) OR
    (stHealth.xConfigurationValid <>
     stPrevious.xConfigurationValid) OR
    (stHealth.uiHighestSeverity <>
     stPrevious.uiHighestSeverity) OR
    (stHealth.uiBlockingReasonCode <>
     stPrevious.uiBlockingReasonCode) OR
    (stHealth.uiDegradedReasonCode <>
     stPrevious.uiDegradedReasonCode);

IF NOT xInitialized THEN
    xInitialized := TRUE;
ELSIF xMaterialChange THEN
    xTransitionEvent := TRUE;
    IF stHealth.udiStatusSequence < 16#FFFFFFFF THEN
        stHealth.udiStatusSequence :=
            stHealth.udiStatusSequence + 1;
    END_IF;
END_IF;

stPrevious := stHealth;

END_FUNCTION_BLOCK

(* ---- FB_IOManager.st ---- *)
FUNCTION_BLOCK FB_IOManager
VAR_INPUT
    stRawInputs : ST_IO;
    xHardwareConfigValid : BOOL;
    xWatchdogHealthy : BOOL;
    stRequestedOutputs : ST_IO;
    xOutputsPermitted : BOOL;
    xSafetyOK : BOOL;
    xCommissioningMode : BOOL;
    udiCommandSequence : UDINT;
END_VAR
VAR_OUTPUT
    stValidatedInputs : ST_IO;
    stAppliedOutputs : ST_IO;
    xReady : BOOL;
    xFault : BOOL;
    uiDiagnosticCode : UINT;
END_VAR
VAR
    xInitialized : BOOL;
    xApplyRequestedOutputs : BOOL;
    iChannel : INT;
END_VAR
VAR CONSTANT
    c_uiDiagnosticNone : UINT := 0;
    c_uiDiagnosticConfigInvalid : UINT := 10;
    c_uiDiagnosticModuleOffline : UINT := 11;
    c_uiDiagnosticWatchdog : UINT := 12;
    c_uiDiagnosticSafetyInhibit : UINT := 13;
    c_uiDiagnosticPermissionInhibit : UINT := 14;
    c_uiDiagnosticForceRejected : UINT := 15;
    c_uiDiagnosticForceConfigurationMissing : UINT := 16;
END_VAR

(* Inputs are copied once to create the immutable application snapshot. *)
FOR iChannel := 0 TO 63 DO
    stValidatedInputs.axDigitalInput[iChannel] := stRawInputs.axDigitalInput[iChannel];
    stValidatedInputs.axDigitalInputValid[iChannel] := stRawInputs.axDigitalInputValid[iChannel];
    stValidatedInputs.axDigitalOutput[iChannel] := FALSE;
    stValidatedInputs.axDigitalOutputValid[iChannel] := FALSE;
END_FOR;

FOR iChannel := 0 TO 15 DO
    stValidatedInputs.adiAnalogInput[iChannel] := stRawInputs.adiAnalogInput[iChannel];
    stValidatedInputs.axAnalogInputValid[iChannel] := stRawInputs.axAnalogInputValid[iChannel];
    stValidatedInputs.adiAnalogOutput[iChannel] := 0;
    stValidatedInputs.axAnalogOutputValid[iChannel] := FALSE;
END_FOR;

stValidatedInputs.xRequiredModulesOnline := stRawInputs.xRequiredModulesOnline;
stValidatedInputs.xForceActive := FALSE;
stValidatedInputs.uiInvalidInputCount := stRawInputs.uiInvalidInputCount;
stValidatedInputs.uiInvalidOutputCount := 0;
stValidatedInputs.uiOutputMismatchCount := 0;

xReady := xHardwareConfigValid AND
          xWatchdogHealthy AND
          stRawInputs.xRequiredModulesOnline;

xFault := NOT xHardwareConfigValid OR
          NOT xWatchdogHealthy OR
          NOT stRawInputs.xRequiredModulesOnline;

xApplyRequestedOutputs := xInitialized AND
                          xReady AND
                          xOutputsPermitted AND
                          xSafetyOK AND
                          NOT stRequestedOutputs.xForceActive;

uiDiagnosticCode := c_uiDiagnosticNone;

IF NOT xHardwareConfigValid THEN
    uiDiagnosticCode := c_uiDiagnosticConfigInvalid;
ELSIF NOT stRawInputs.xRequiredModulesOnline THEN
    uiDiagnosticCode := c_uiDiagnosticModuleOffline;
ELSIF NOT xWatchdogHealthy THEN
    uiDiagnosticCode := c_uiDiagnosticWatchdog;
ELSIF NOT xSafetyOK THEN
    uiDiagnosticCode := c_uiDiagnosticSafetyInhibit;
ELSIF NOT xOutputsPermitted THEN
    uiDiagnosticCode := c_uiDiagnosticPermissionInhibit;
ELSIF stRequestedOutputs.xForceActive THEN
    IF xCommissioningMode THEN
        uiDiagnosticCode := c_uiDiagnosticForceConfigurationMissing;
    ELSE
        uiDiagnosticCode := c_uiDiagnosticForceRejected;
    END_IF;
END_IF;

(* FALSE and zero are the current approved baseline safe image.
   A future non-zero safe channel requires an approved IO configuration. *)
FOR iChannel := 0 TO 63 DO
    stAppliedOutputs.axDigitalInput[iChannel] :=
        stValidatedInputs.axDigitalInput[iChannel];
    stAppliedOutputs.axDigitalInputValid[iChannel] :=
        stValidatedInputs.axDigitalInputValid[iChannel];
    stAppliedOutputs.axDigitalOutputValid[iChannel] :=
        stRequestedOutputs.axDigitalOutputValid[iChannel] AND xHardwareConfigValid;

    IF xApplyRequestedOutputs AND
       stRequestedOutputs.axDigitalOutputValid[iChannel] THEN
        stAppliedOutputs.axDigitalOutput[iChannel] :=
            stRequestedOutputs.axDigitalOutput[iChannel];
    ELSE
        stAppliedOutputs.axDigitalOutput[iChannel] := FALSE;
    END_IF;
END_FOR;

FOR iChannel := 0 TO 15 DO
    stAppliedOutputs.adiAnalogInput[iChannel] :=
        stValidatedInputs.adiAnalogInput[iChannel];
    stAppliedOutputs.axAnalogInputValid[iChannel] :=
        stValidatedInputs.axAnalogInputValid[iChannel];
    stAppliedOutputs.axAnalogOutputValid[iChannel] :=
        stRequestedOutputs.axAnalogOutputValid[iChannel] AND xHardwareConfigValid;

    IF xApplyRequestedOutputs AND
       stRequestedOutputs.axAnalogOutputValid[iChannel] THEN
        stAppliedOutputs.adiAnalogOutput[iChannel] :=
            stRequestedOutputs.adiAnalogOutput[iChannel];
    ELSE
        stAppliedOutputs.adiAnalogOutput[iChannel] := 0;
    END_IF;
END_FOR;

stAppliedOutputs.xRequiredModulesOnline := stRawInputs.xRequiredModulesOnline;
stAppliedOutputs.xForceActive := FALSE;
stAppliedOutputs.uiInvalidInputCount := stRawInputs.uiInvalidInputCount;
stAppliedOutputs.uiInvalidOutputCount := stRequestedOutputs.uiInvalidOutputCount;
stAppliedOutputs.uiOutputMismatchCount := 0;
stAppliedOutputs.uiDiagnosticCode := uiDiagnosticCode;

IF stAppliedOutputs.udiImageSequence < c_udiCounterMaximum THEN
    stAppliedOutputs.udiImageSequence :=
        stAppliedOutputs.udiImageSequence + 1;
END_IF;

stValidatedInputs.udiImageSequence := stAppliedOutputs.udiImageSequence;
stValidatedInputs.uiDiagnosticCode := uiDiagnosticCode;

xInitialized := TRUE;

END_FUNCTION_BLOCK
